(* Logix 5000 project; controller capstone_rev_1 Emulate 5570 rev 35.11; software revision 35.01 *)

TASK MainTask (continuous, watchdog 500 ms) : MainProgram

MODULES
   Local : Emulate 5570 (ICP 0, rev 35.11)
END_MODULES

PROGRAM MainProgram   (* main routine MainRoutine *)
VAR
   Analog_Input : REAL;
   Auto_Select : BOOL;
   Decarbonization_Area : BOOL;
   Decarbonization_Pump : BOOL;
   Decarbonization_Pump_PB : BOOL;
   Decarbonization_Temp : BOOL;
   Decarbonization_Timer : TIMER := (PRE := 1200000);
   Decarbonization_Valve : BOOL;
   Decarbonization_Valve_PB : BOOL;
   Down_Limit_Switch : BOOL;
   Drying_Area : BOOL;
   Drying_Timer : TIMER := (PRE := 180000);
   Encoder : REAL;
   Encoder_Analog_Input : REAL;
   Fan1 : BOOL;
   Fan2 : BOOL;
   Fan_PB : BOOL;
   Heater : BOOL;
   Heater_Switch : BOOL;
   High_Lvl_Sensor : BOOL;
   Hoist_Down : BOOL;
   Hoist_Down_PB : BOOL;
   Hoist_Fwd : BOOL;
   Hoist_Fwd_PB : BOOL;
   Hoist_Rev : BOOL;
   Hoist_Rev_PB : BOOL;
   Hoist_Up : BOOL;
   Hoist_Up_PB : BOOL;
   Home_PB : BOOL;
   Home_Position : BOOL;
   Low_Lvl_Sensor : BOOL;
   Manual_Select : BOOL;
   Offloading_Area : BOOL;
   Position : SCALE;
   Process_Counter : COUNTER := (PRE := 10);
   Process_Done_Timer : TIMER := (PRE := 2000);
   Process_Start_Timer : TIMER := (PRE := 3000);
   Pulse : BOOL;
   Rack_in_Decarbonization : BOOL;
   Rack_in_Drying : BOOL;
   Rack_in_Loading_Area : BOOL;
   Rack_in_Wrinsing : BOOL;
   Rack_Scale : BOOL;
   Reset_PB : BOOL;
   Temp_OK : BOOL;
   Temp_Sensor : REAL;
   Temperature : SCALE;
   Up_Limit_Switch : BOOL;
   Weighing_Scale : DINT;
   Wrinsing_Area : BOOL;
   Wrinsing_Pump : BOOL;
   Wrinsing_Pump_PB : BOOL;
   Wrinsing_Timer : TIMER := (PRE := 120000);
END_VAR

ROUTINE Analog_Routine   (* ladder *)
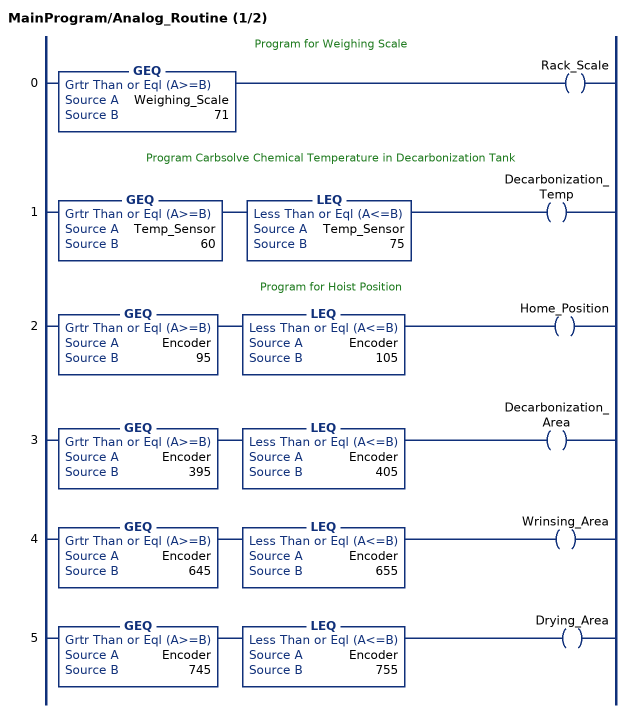
   // Program for Weighing Scale
   0: GEQ(Weighing_Scale,71)OTE(Rack_Scale);
   // Program Carbsolve Chemical Temperature in Decarbonization Tank
   1: GEQ(Temp_Sensor,60)LEQ(Temp_Sensor,75)OTE(Decarbonization_Temp);
   // Program for Hoist Position
   2: GEQ(Encoder,95)LEQ(Encoder,105)OTE(Home_Position);
   3: GEQ(Encoder,395)LEQ(Encoder,405)OTE(Decarbonization_Area);
   4: GEQ(Encoder,645)LEQ(Encoder,655)OTE(Wrinsing_Area);
   5: GEQ(Encoder,745)LEQ(Encoder,755)OTE(Drying_Area);
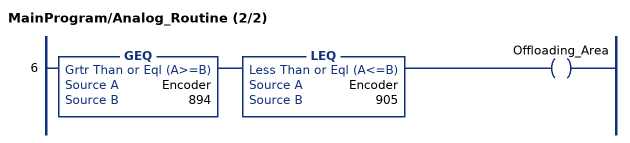
   6: GEQ(Encoder,894)LEQ(Encoder,905)OTE(Offloading_Area);
END_ROUTINE

ROUTINE MainRoutine   (* ladder *)
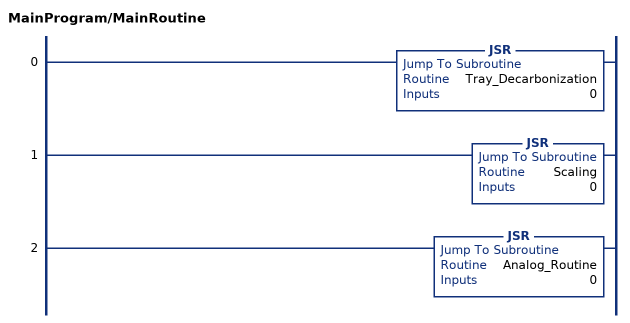
   0: JSR(Tray_Decarbonization,0);
   1: JSR(Scaling,0);
   2: JSR(Analog_Routine,0);
END_ROUTINE

ROUTINE Scaling   (* function block diagram *)
   SHEET 1
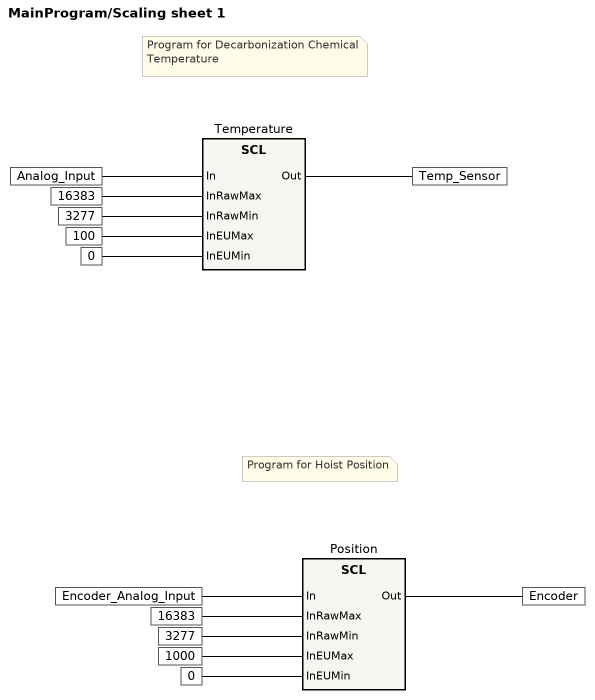
   // Program for Decarbonization Chemical
   // Temperature
   Temperature : SCL(In := Analog_Input, InRawMax := 16383, InRawMin := 3277, InEUMax := 100, InEUMin := 0);
   // Program for Hoist Position
   Position : SCL(In := Encoder_Analog_Input, InRawMax := 16383, InRawMin := 3277, InEUMax := 1000, InEUMin := 0);
   Temp_Sensor := Temperature.Out;
   Encoder := Position.Out;
END_ROUTINE

ROUTINE Tray_Decarbonization   (* ladder *)
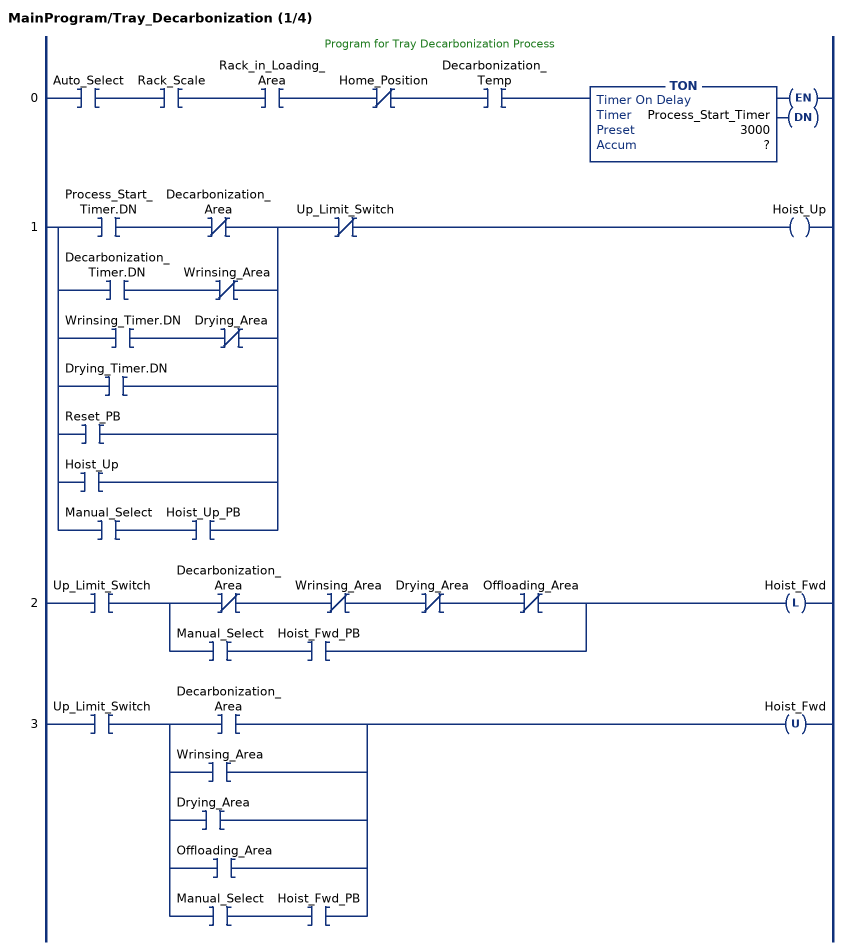
   // Program for Tray Decarbonization Process
   0: XIC(Auto_Select)XIC(Rack_Scale)XIC(Rack_in_Loading_Area)XIO(Home_Position)XIC(Decarbonization_Temp)TON(Process_Start_Timer,?,?);
   1: [XIC(Process_Start_Timer.DN) XIO(Decarbonization_Area) ,XIC(Decarbonization_Timer.DN) XIO(Wrinsing_Area) ,XIC(Wrinsing_Timer.DN) XIO(Drying_Area) ,XIC(Drying_Timer.DN) ,[XIC(Reset_PB) ,XIC(Hoist_Up) ] ,XIC(Manual_Select) XIC(Hoist_Up_PB) ]XIO(Up_Limit_Switch)OTE(Hoist_Up);
   2: XIC(Up_Limit_Switch)[XIO(Decarbonization_Area) XIO(Wrinsing_Area) XIO(Drying_Area) XIO(Offloading_Area) ,XIC(Manual_Select) XIC(Hoist_Fwd_PB) ]OTL(Hoist_Fwd);
   3: XIC(Up_Limit_Switch)[XIC(Decarbonization_Area) ,XIC(Wrinsing_Area) ,XIC(Drying_Area) ,XIC(Offloading_Area) ,XIC(Manual_Select) XIC(Hoist_Fwd_PB) ]OTU(Hoist_Fwd);
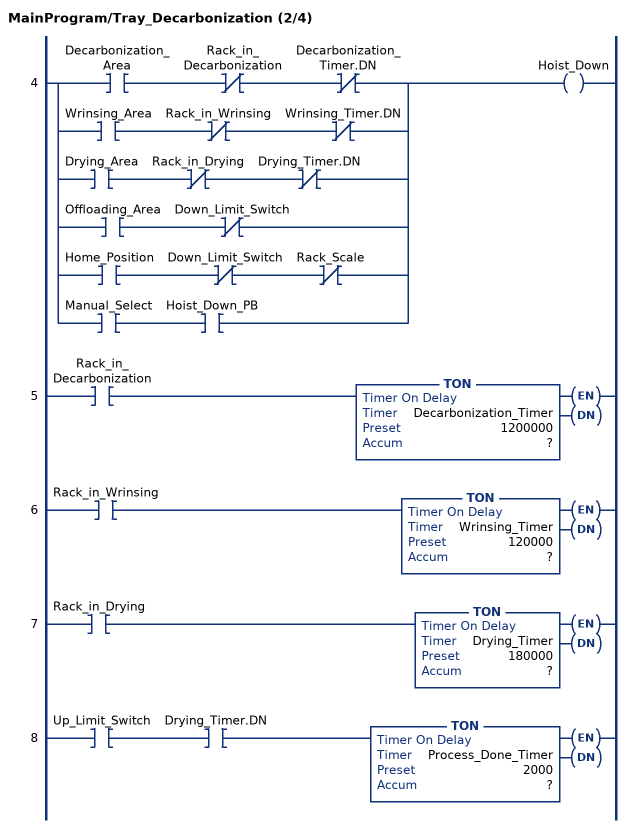
   4: [XIC(Decarbonization_Area) XIO(Rack_in_Decarbonization) XIO(Decarbonization_Timer.DN) ,XIC(Wrinsing_Area) XIO(Rack_in_Wrinsing) XIO(Wrinsing_Timer.DN) ,XIC(Drying_Area) XIO(Rack_in_Drying) XIO(Drying_Timer.DN) ,XIC(Offloading_Area) XIO(Down_Limit_Switch) ,XIC(Home_Position) XIO(Down_Limit_Switch) XIO(Rack_Scale) ,XIC(Manual_Select) XIC(Hoist_Down_PB) ]OTE(Hoist_Down);
   5: XIC(Rack_in_Decarbonization)TON(Decarbonization_Timer,?,?);
   6: XIC(Rack_in_Wrinsing)TON(Wrinsing_Timer,?,?);
   7: XIC(Rack_in_Drying)TON(Drying_Timer,?,?);
   8: XIC(Up_Limit_Switch)XIC(Drying_Timer.DN)TON(Process_Done_Timer,?,?);
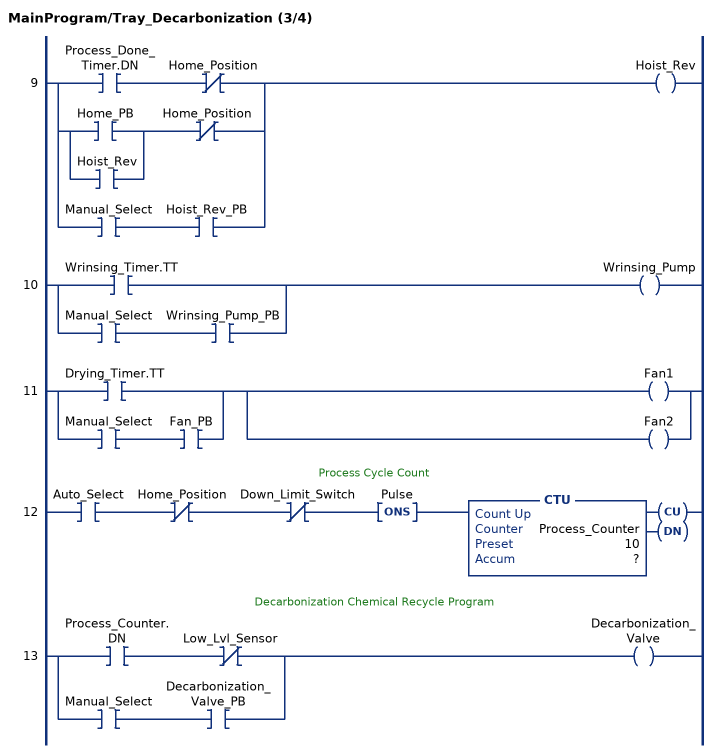
   9: [XIC(Process_Done_Timer.DN) XIO(Home_Position) ,[XIC(Home_PB) ,XIC(Hoist_Rev) ] XIO(Home_Position) ,XIC(Manual_Select) XIC(Hoist_Rev_PB) ]OTE(Hoist_Rev);
   10: [XIC(Wrinsing_Timer.TT) ,XIC(Manual_Select) XIC(Wrinsing_Pump_PB) ]OTE(Wrinsing_Pump);
   11: [XIC(Drying_Timer.TT) ,XIC(Manual_Select) XIC(Fan_PB) ][OTE(Fan1) ,OTE(Fan2) ];
   // Process Cycle Count
   12: XIC(Auto_Select)XIO(Home_Position)XIO(Down_Limit_Switch)ONS(Pulse)CTU(Process_Counter,?,?);
   // Decarbonization Chemical Recycle Program
   13: [XIC(Process_Counter.DN) XIO(Low_Lvl_Sensor) ,XIC(Manual_Select) XIC(Decarbonization_Valve_PB) ]OTE(Decarbonization_Valve);
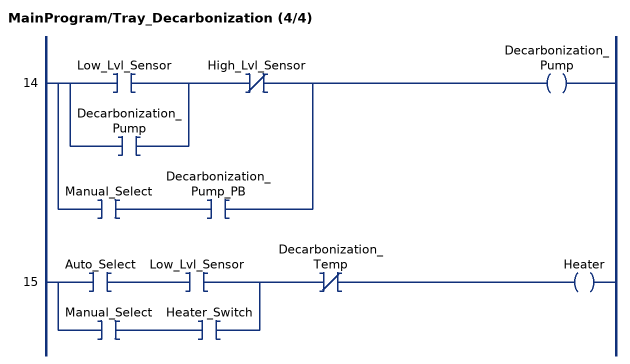
   14: [[XIC(Low_Lvl_Sensor) ,XIC(Decarbonization_Pump) ] XIO(High_Lvl_Sensor) ,XIC(Manual_Select) XIC(Decarbonization_Pump_PB) ]OTE(Decarbonization_Pump);
   15: [XIC(Auto_Select) XIC(Low_Lvl_Sensor) ,XIC(Manual_Select) XIC(Heater_Switch) ]XIO(Decarbonization_Temp)OTE(Heater);
END_ROUTINE
END_PROGRAM
